Fanuc KAREL source: kt00935.compact.KL

PROGRAM KT00935
%STACKSIZE=65535
%PRIORITY=65535
%NOLOCKGROUP
VAR
ENTRY : INTEGER
PNAME : STRING[80]
VNAME : STRING[80]
STATUS : INTEGER
VALUE : BOOLEAN
BEGIN
ENTRY=0
PNAME=''
VNAME='VALUE'
GET_VAR(ENTRY,PNAME,VNAME,VALUE,STATUS)
END KT00935
